(* IEC 61131-3 sources: eCockpitGit/test_project/src/%F%00 Library/%F%Common Functions/%F%String/%F%Big Input/%F%Edit, 5 files *)

(* ---- %POU%FU_sDeleteBI.st ---- *)
// +-----------+----------+----------+-----------------------------------------------------------------------------------------------------------------------+
// |**Version**|**Author**| **Date** |**Changes**                                                                                                            |
// +-----------+----------+----------+-----------------------------------------------------------------------------------------------------------------------+
// | 1         | NSN      | 13-06-18 | Creation                                                                                                              |
// +-----------+----------+----------+-----------------------------------------------------------------------------------------------------------------------+
// | 1.1       | NSN      | 05-02-19 | Made dependant on big output version                                                                                  |
// +-----------+----------+----------+-----------------------------------------------------------------------------------------------------------------------+
FUNCTION FU_sDeleteBI : STRING(255)
VAR_IN_OUT
	sStr		:STRING(1);			//Input String
END_VAR
VAR_INPUT
	wLen		:WORD;				//Amount to delete
	wPos		:WORD;				//Position to delete from
END_VAR
(*%!%__DELIMITER__%!%*)
FU_sDeleteBIBO(sOut:= FU_sDeleteBI,sStr:= sStr,wLen:= wLen,wPos:= wPos,wOutSize:= 255);

(* ---- %POU%FU_sDeleteRightBI.st ---- *)
//This functions deletes a part of a string values are counted from the right instead of the left
// +-----------+----------+----------+-----------------------------------------------------------------------------------------------------------------------+
// |**Version**|**Author**| **Date** |**Changes**                                                                                                            |
// +-----------+----------+----------+-----------------------------------------------------------------------------------------------------------------------+
// | 1         | NSN      | 22-02-19 | Creation                                                                                                              |
// +-----------+----------+----------+-----------------------------------------------------------------------------------------------------------------------+
FUNCTION FU_sDeleteRightBI : STRING(255)
VAR_IN_OUT
	sStr		:STRING(1);			//Input String
END_VAR
VAR_INPUT
	wLen		:WORD;				//Amount to trim from end
	wPos		:WORD;				//Position to delete from
END_VAR
(*%!%__DELIMITER__%!%*)
FU_sDeleteRightBIBO(sOut:= FU_sDeleteRightBI, sStr:= sStr, wLen:= wLen,wPos:= wPos, wOutSize:= 255);

(* ---- %POU%FU_sMidBI.st ---- *)
//This functions extracts a part of a string
// |**Version**|**Author**| **Date** |**Changes**
// | 1         | NSN      | 13-06-18 | Creation                                                                                                              |
// | 1.1       | NSN      | 05-02-19 | Made dependant on big output version                                                                                  |
FUNCTION FU_sMidBI : STRING(255)
VAR_IN_OUT
	sStr		:STRING(1);			//Input String
END_VAR
VAR_INPUT
	wLen		:WORD;				//Amount to copy
	wPos		:WORD;				//Position to copy from
END_VAR
(*%!%__DELIMITER__%!%*)
FU_sMidBIBO(sOut:= FU_sMidBI,sStr:= sStr,wLen:= wLen,wPos:= wPos,wOutSize:= 255);

(* ---- %POU%FU_sMidRightBI.st ---- *)
//This functions extracts a part of a string, values are counted from the right instead of the left
// +-----------+----------+----------+-----------------------------------------------------------------------------------------------------------------------+
// |**Version**|**Author**| **Date** |**Changes**                                                                                                            |
// +-----------+----------+----------+-----------------------------------------------------------------------------------------------------------------------+
// | 1         | NSN      | 22-02-19 | Creation                                                                                                              |
// +-----------+----------+----------+-----------------------------------------------------------------------------------------------------------------------+
FUNCTION FU_sMidRightBI : STRING(255)
VAR_IN_OUT
	sStr		:STRING(1);			//Input String
END_VAR
VAR_INPUT
	wLen		:WORD;				//Amount to copy
	wPos		:WORD;				//Position to copy from
END_VAR
(*%!%__DELIMITER__%!%*)
FU_sMidRightBIBO(sOut:= FU_sMidRightBI,sStr:= sStr,wLen:= wLen,wPos:= wPos,wOutSize:= 255);

(* ---- %POU%FU_sReplaceCharBI.st ---- *)
//This functions replaces all instances of a character with another
// |**Version**|**Author**| **Date** |**Changes**
// | 1         | NSN      | 13-06-18 | Creation                                                                                                              |
FUNCTION FU_sReplaceCharBI
VAR_IN_OUT
	str			:STRING(1);			//Input String
END_VAR
VAR_INPUT
	eOGChar		:EASCII;				//Character to replace
	eReplaceChar:EASCII;				//Character to replace by
END_VAR
VAR
	pStr		:POINTER TO BYTE;	//Address of the string
END_VAR
(*%!%__DELIMITER__%!%*)
pStr					:=		ADR(str);
WHILE pStr^ <> 0 DO
	IF pStr^ = eOGChar THEN
		pStr^			:=		eReplaceChar;
	END_IF
	pStr				:=		pStr + 1;
END_WHILE
